FUNCTION_BLOCK L2_Cinta_SFC  EXTENDS L1_ControllerBase_SFC

VAR_INPUT 					// Sensores y comandos
	Situar		: BOOL;
	Transferir	: BOOL;	
	pp			: BOOL; 	// presencia de pale
	cp0			: BOOL;
	cp1			: BOOL;
	cp2			: BOOL;
END_VAR

VAR_OUTPUT					// Actuadores
	RUN			: BOOL; 	// activa motor
	REV			: BOOL; 	// invierte motor
	R_1			: BOOL; 	// retenedor baja
	S_1			: BOOL; 	// separador sube
END_VAR

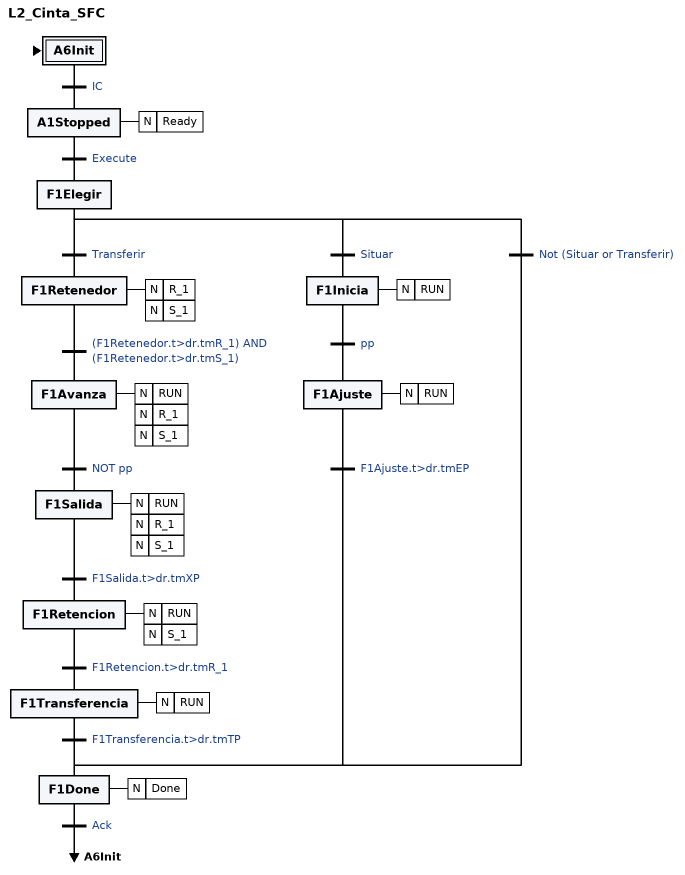
INITIAL_STEP A6Init:
END_STEP
TRANSITION FROM A6Init TO A1Stopped
    := IC;
END_TRANSITION
STEP A1Stopped:
    Ready(N);
END_STEP
TRANSITION FROM A1Stopped TO F1Elegir
    := Execute;
END_TRANSITION
STEP F1Elegir:
END_STEP
TRANSITION FROM F1Elegir TO F1Retenedor
    := Transferir;
END_TRANSITION
STEP F1Retenedor:
    R_1(N);
    S_1(N);
END_STEP
TRANSITION FROM F1Retenedor TO F1Avanza
    := (F1Retenedor.t>dr.tmR_1) AND (F1Retenedor.t>dr.tmS_1);
END_TRANSITION
STEP F1Avanza:
    RUN(N);
    R_1(N);
    S_1(N);
END_STEP
TRANSITION FROM F1Avanza TO F1Salida
    := NOT pp;
END_TRANSITION
STEP F1Salida:
    RUN(N);
    R_1(N);
    S_1(N);
END_STEP
TRANSITION FROM F1Salida TO F1Retencion
    := F1Salida.t>dr.tmXP;
END_TRANSITION
STEP F1Retencion:
    RUN(N);
    S_1(N);
END_STEP
TRANSITION FROM F1Retencion TO F1Transferencia
    := F1Retencion.t>dr.tmR_1;
END_TRANSITION
STEP F1Transferencia:
    RUN(N);
END_STEP
TRANSITION FROM F1Transferencia TO F1Done
    := F1Transferencia.t>dr.tmTP;
END_TRANSITION
TRANSITION FROM F1Elegir TO F1Inicia
    := Situar;
END_TRANSITION
STEP F1Inicia:
    RUN(N);
END_STEP
TRANSITION FROM F1Inicia TO F1Ajuste
    := pp;
END_TRANSITION
STEP F1Ajuste:
    RUN(N);
END_STEP
TRANSITION FROM F1Ajuste TO F1Done
    := F1Ajuste.t>dr.tmEP;
END_TRANSITION
TRANSITION FROM F1Elegir TO F1Done
    := Not (Situar or Transferir);
END_TRANSITION
STEP F1Done:
    Done(N);
END_STEP
TRANSITION FROM F1Done TO A6Init
    := Ack;
END_TRANSITION

END_FUNCTION_BLOCK

(* stored: Version 1.1.0.1, ProductVersion 3.1.4024.11
   POU L2_Cinta_SFC: Id {7a4e0e2e-bc1d-4eb2-80cf-952f4dd5e6da}, SpecialFunc None *)
